// TIA Portal V16 export
// export: Created 2024-09-05T17:39:18.4673265Z, ExportSetting WithDefaults, DisplayName Totally Integrated Automation Portal, DisplayVersion V16 Update 6, DisplayName TIA Portal Version Control Interface, DisplayVersion V16 Update 2, DisplayName TIA Portal Openness, DisplayVersion V16 Update 6, DisplayName STEP 7 Professional, DisplayVersion V16 Update 6, DisplayName STEP 7 Safety, DisplayVersion V16, DisplayName WinCC Advanced, DisplayVersion V16 Update 6
DATA_BLOCK "AutoPositions"   // DB11
{ S7_Optimized_Access := 'TRUE' }
VERSION : 0.1
// stored: AutoNumber true, DBAccessibleFromOPCUA true, IsOnlyStoredInLoadMemory false, IsRetainMemResEnabled false, IsWriteProtectedInAS false, MemoryReserve 100
   VAR RETAIN
      St1_Table1 : "UDT_PositionData";
      St2_Table2 : "UDT_PositionData";
      St3_Fitting : "UDT_PositionData";
      R1_Gripper : "UDT_PositionData";
      AE_Gripper : "UDT_PositionData";
      St4_OKposition : "UDT_PositionData";
   END_VAR
   VAR
      emptyPos : "UDT_PositionData";
   END_VAR
BEGIN
END_DATA_BLOCK
